(* CoDeSys 2.3.9.37 project: tranvia.pro *)
(* Libraries: Standard.lib 4.10.05 12:14:46, IecSfc.lib 13.4.06 16:51:28 *)

(* Global variable list: Global_Variables *)
VAR_GLOBAL

   (*Entradas*)
   S1 : BOOL;
   S2:BOOL;

   (* Salidas *)
   Sem1CRojo:BOOL ;
   Sem1CAmbar:BOOL;
   Sem1CVerde:BOOL ;
   Sem1PRojo:BOOL ;
   Sem1PVerde:BOOL ;

END_VAR

(* POU PLC_PRG, ST *)
PROGRAM PLC_PRG
VAR
END_VAR
Visualizacion;
END_PROGRAM

(* POU Visualizacion, ST *)
PROGRAM Visualizacion
VAR
   posx: INT :=0;
   posy: INT:= 0;
   ang:INT :=20;
   vectorx : ARRAY[1..56] OF INT :=0,-10,-20,-30,-40,-50,-60,-70,-80,-90,-100,-110,-120,-130,-140,-150,-160,-170,-190,-210,-230,-250,-270,-290,-310,-330,-350,-370,-390,-410,-430,-450,-470,-490,-510,-530,-550,-570,-590,-610,-620,-630,-640,-650,-660,-670,-680,-690,-700,-710,-720,-730,-740,-750,-760,-770;
   vectory : ARRAY[1..56] OF INT:= 21,19,16,10,6,2,-2,-5,-12,-14,-18,-24,-27,-33,-38,-43,-51,-61,-73,-87,-102,-118,-134,-149,-163,-176,-190,-200,-208,-214,-221,-222,-223,-218,-218,-214,-210,-208,-204,-199,-194,-194,-193,-189,-189,-186,-186,-186,-186,-186,-186,-186,-186,-186,-186,-186;
   vectorang : ARRAY[1..56] OF INT:= 220,20,20,20,20,22,22,22,24,25,27,29,30,32,34,35,35,35,37,37,37,37,37,37,34,32,28,24,19,13,4,0,-6,-9,-11,-13,-13,-13,-11,-8,-8,-8,-5,-4,-4,0,0,0,0,0,0,0,0,0,0,0;
   i: INT :=1;

	trenizq: BOOL;
	BotonIzq: BOOL;
	BotonDer: BOOL;
	trender: BOOL;
      cont_vel:INT;
      factor_vel:INT :=1;
	cambiaindice: BOOL;
END_VAR
IF NOT trenizq AND NOT trender THEN
   posx:=10000;
   posy:=10000;
END_IF

IF BotonIzq THEN
   trenizq:=TRUE;
   i:=56;
END_IF

IF BotonDer THEN
   trender:=TRUE;
   i:=1;
END_IF


(*Velocidad del tranvia *)
IF (trenizq OR trender) THEN
  IF  cont_vel=factor_vel THEN
     cont_vel:=1;
     cambiaindice:=TRUE;
  ELSE
     cont_vel:=cont_vel+1;;
     cambiaindice:=FALSE;
 END_IF
END_IF


IF trenizq THEN
   posx:=vectorx[i];
   posy:=vectory[i];
   ang:=vectorang[i];
   IF cambiaindice THEN
         i:=i-1;
   END_IF;
   IF i=0 THEN
      trenizq:=FALSE;
  END_IF
END_IF



IF trender THEN
   posx:=vectorx[i];
   posy:=vectory[i];
   ang:=vectorang[i];
  IF cambiaindice THEN
      i:=i+1;
  END_IF
   IF i=57 THEN
      trender:=FALSE;
  END_IF
END_IF



IF i>=5 AND i<=17 THEN
   S2:=TRUE;
ELSE
   S2:=FALSE;
END_IF;

IF i>=40 AND i<=54 THEN
   S1:=TRUE;
ELSE
   S1:=FALSE;
END_IF;
END_PROGRAM

(* Visualisation Visu
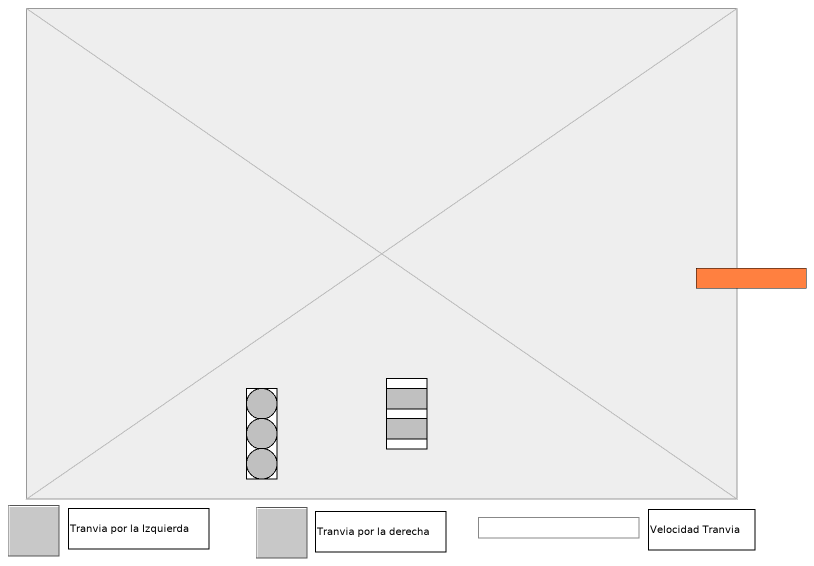
bitmap at (60,30)-(771,521): C:\USERS\USUARIO\DROPBOX\AUTOMATIZACION INDUSTRIAL\APUNTES\TRANVIA.BMP
polygon at (730,290)-(840,310): x offset Visualizacion.posx; y offset Visualizacion.posy; angle Visualizacion.ang
button at (42,527)-(93,578): taps Visualizacion.BotonIzq
button at (290,529)-(341,580): taps Visualizacion.BotonDer
rectangle at (102,530)-(243,571): text "Tranvia por la Izquierda"
rectangle at (349,533)-(480,574): text "Tranvia por la derecha"
rectangle at (682,531)-(789,572): text "Velocidad Tranvia"
ellipse at (280,410)-(311,441): alarm colour if Sem1CRojo
ellipse at (280,440)-(311,471): alarm colour if Sem1CAmbar
ellipse at (280,470)-(311,501): alarm colour if Sem1CVerde
rounded rectangle at (420,410)-(461,431): alarm colour if Sem1PRojo
rounded rectangle at (420,440)-(461,461): alarm colour if Sem1Pverde
3 more shapes without text or variables
*)
